{attribute 'qualified_only'}
{attribute 'strict'}
{attribute 'to_string'}
TYPE E_CurrentState :
(
	Init,
	GalvoHandling,
	MirrorAdj,
	FinishedProduct

);
END_TYPE

(* stored: Version 1.1.0.1
   DUT E_CurrentState: Id {9732b89e-9199-44b0-a0ce-f51206418553} *)
